FUNCTION_BLOCK xPPU_Crane
VAR_INPUT
	i_error: POINTER TO ErrorManager;
	i_process: POINTER TO ProcessManager;
	i_state: POINTER TO StateTracker;
END_VAR
VAR
	m_emptyParams: ParameterSet;
	m_subRes: EOperationResult;
	m_alarm_flags: ARRAY [1..10] OF BOOL := [FALSE, FALSE, FALSE, FALSE, FALSE, FALSE,FALSE, FALSE, FALSE, FALSE]; 
	m_timer_LSC_EntryCheck : TON;
END_VAR

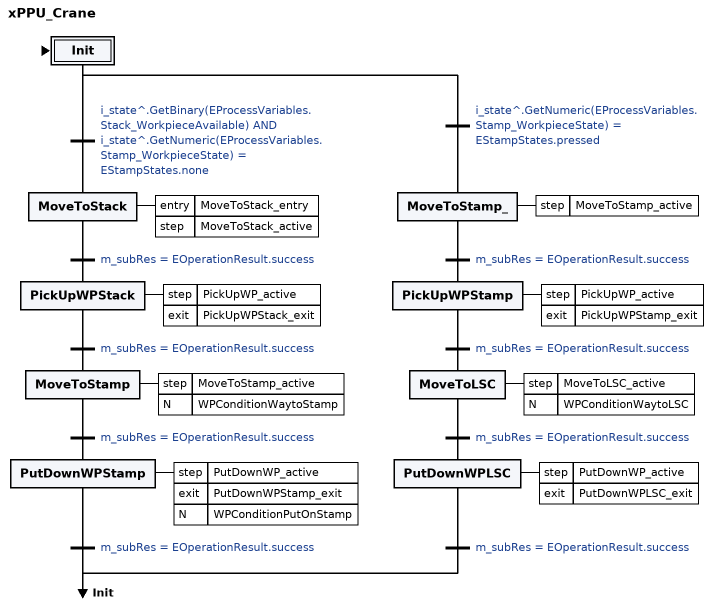
INITIAL_STEP Init:
END_STEP
TRANSITION FROM Init TO MoveToStack
    := i_state^.GetBinary(EProcessVariables.Stack_WorkpieceAvailable) AND i_state^.GetNumeric(EProcessVariables.Stamp_WorkpieceState) = EStampStates.none;
END_TRANSITION
STEP MoveToStack:
    MoveToStack_entry(P1);  // entry action
    MoveToStack_active(N);  // step action
END_STEP
TRANSITION FROM MoveToStack TO PickUpWPStack
    := m_subRes = EOperationResult.success;
END_TRANSITION
STEP PickUpWPStack:
    PickUpWP_active(N);  // step action
    PickUpWPStack_exit(P0);  // exit action
END_STEP
TRANSITION FROM PickUpWPStack TO MoveToStamp
    := m_subRes = EOperationResult.success;
END_TRANSITION
STEP MoveToStamp:
    MoveToStamp_active(N);  // step action
    WPConditionWaytoStamp(N);
END_STEP
TRANSITION FROM MoveToStamp TO PutDownWPStamp
    := m_subRes = EOperationResult.success;
END_TRANSITION
STEP PutDownWPStamp:
    PutDownWP_active(N);  // step action
    PutDownWPStamp_exit(P0);  // exit action
    WPConditionPutOnStamp(N);
END_STEP
TRANSITION FROM PutDownWPStamp TO Init
    := m_subRes = EOperationResult.success;
END_TRANSITION
TRANSITION FROM Init TO MoveToStamp_
    := i_state^.GetNumeric(EProcessVariables.Stamp_WorkpieceState) = EStampStates.pressed;
END_TRANSITION
STEP MoveToStamp_:
    MoveToStamp_active(N);  // step action
END_STEP
TRANSITION FROM MoveToStamp_ TO PickUpWPStamp
    := m_subRes = EOperationResult.success;
END_TRANSITION
STEP PickUpWPStamp:
    PickUpWP_active(N);  // step action
    PickUpWPStamp_exit(P0);  // exit action
END_STEP
TRANSITION FROM PickUpWPStamp TO MoveToLSC
    := m_subRes = EOperationResult.success;
END_TRANSITION
STEP MoveToLSC:
    MoveToLSC_active(N);  // step action
    WPConditionWaytoLSC(N);
END_STEP
TRANSITION FROM MoveToLSC TO PutDownWPLSC
    := m_subRes = EOperationResult.success;
END_TRANSITION
STEP PutDownWPLSC:
    PutDownWP_active(N);  // step action
    PutDownWPLSC_exit(P0);  // exit action
END_STEP
TRANSITION FROM PutDownWPLSC TO Init
    := m_subRes = EOperationResult.success;
END_TRANSITION

ACTION MoveToLSC_active:
m_subRes := i_process^.Execute(
	EBehaviorType.control_primitive,
	EPrimitives.Crane_MoveToLSC,
	m_emptyParams);
END_ACTION

ACTION MoveToStack_active:
m_subRes := i_process^.Execute(
	EBehaviorType.control_primitive,
	EPrimitives.Crane_MoveToStack,
	m_emptyParams);
END_ACTION

ACTION MoveToStack_entry:

END_ACTION

ACTION MoveToStamp_active:
m_subRes := i_process^.Execute(
	EBehaviorType.control_primitive,
	EPrimitives.Crane_MoveToStamp,
	m_emptyParams);
END_ACTION

ACTION PickUpWP_active:
m_subRes := i_process^.Execute(
	EBehaviorType.control_primitive,
	EPrimitives.Crane_PickUpWP,
	m_emptyParams);
END_ACTION

ACTION PickUpWPStack_exit:
i_state^.ShiftProduct(EProducts.stack_product, EProducts.crane_product); 
IF m_alarm_flags[1] = FALSE
	AND i_state^.GetBinary(EProcessVariables.Crane_AtStack)
    AND i_state^.GetBinary(EProcessVariables.Stack_WorkpieceAvailable)
    AND NOT i_state^.GetBinary(EProcessVariables.Crane_HoldingWorkpiece)
THEN 
    i_error^.AddMessage(EAlarms.crane_gripper_failed_stack, TRUE, ESeverity.error, 'Crane failed to pick up the WP at Stack');
    m_alarm_flags[1] := TRUE;
END_IF

IF m_alarm_flags[2] = FALSE
	AND i_state^.GetBinary(EProcessVariables.Crane_AtStack)
    AND NOT i_state^.GetBinary(EProcessVariables.Stack_WorkpieceAvailable) 
    AND NOT i_state^.GetBinary(EProcessVariables.Crane_HoldingWorkpiece)
THEN 
    i_error^.AddMessage(EAlarms.crane_dropped_WP_stack, TRUE, ESeverity.error, 'WP dropped from Crane at Stack');
    m_alarm_flags[2] := TRUE;
END_IF
END_ACTION

ACTION PickUpWPStamp_exit:
i_state^.ShiftProduct(EProducts.stamp_product, EProducts.crane_product);
IF m_alarm_flags[5] = FALSE
    AND i_state^.GetBinary(EProcessVariables.Crane_AtStamp) 
    AND NOT i_state^.GetBinary(EProcessVariables.Crane_HoldingWorkpiece)
	AND i_state^.GetBinary(EProcessVariables.Stamp_WPAtStamp)
THEN 
    i_error^.AddMessage(EAlarms.crane_gripper_failed_stamp, TRUE, ESeverity.error, 'Crane failed pick the WP up at Stamp');
    m_alarm_flags[5] := TRUE;
END_IF

IF m_alarm_flags[6] = FALSE
    AND i_state^.GetBinary(EProcessVariables.Crane_AtStamp) 
    AND NOT i_state^.GetBinary(EProcessVariables.Crane_HoldingWorkpiece)
	AND NOT i_state^.GetBinary(EProcessVariables.Stamp_WPAtStamp)
THEN 
    i_error^.AddMessage(EAlarms.crane_dropped_WP_stamp, TRUE, ESeverity.error, 'WP dropped from Crane at Stamp');
    m_alarm_flags[6] := TRUE;
END_IF
END_ACTION

ACTION PutDownWP_active:
m_subRes := i_process^.Execute(
	EBehaviorType.control_primitive,
	EPrimitives.Crane_PutDownWP,
	m_emptyParams);
END_ACTION

ACTION PutDownWPLSC_exit:
i_state^.ShiftProduct(EProducts.crane_product, EProducts.LSC_product);
END_ACTION

ACTION PutDownWPStamp_exit:
i_state^.ShiftProduct(EProducts.crane_product, EProducts.stamp_product);
END_ACTION

ACTION WPConditionPutOnStamp:
IF m_alarm_flags[4] = FALSE
	AND i_state^.Getbinary(EProcessVariables.Crane_AtStamp)
    AND i_state^.Getbinary(EProcessVariables.Crane_CylinderExtended)
	AND NOT i_state^.Getbinary(EProcessVariables.Stamp_WPAtStamp)
THEN 
    i_error^.AddMessage(EAlarms.crane_putdown_failed_stamp, TRUE, ESeverity.error, 'WP not corrcetly put by the Crane at Stamp');
    m_alarm_flags[4] := TRUE;
END_IF
END_ACTION

ACTION WPConditionWaytoLSC:
IF m_alarm_flags[7] = FALSE
    AND NOT i_state^.GetBinary(EProcessVariables.Crane_HoldingWorkpiece)
THEN 
    i_error^.AddMessage(EAlarms.crane_dropped_WP_WayToLSC, TRUE, ESeverity.error, 'WP dropped from Crane on the way to LSC');
    m_alarm_flags[7] := TRUE;
END_IF
END_ACTION

ACTION WPConditionWaytoStamp:
IF m_alarm_flags[3] = FALSE
    AND NOT i_state^.GetBinary(EProcessVariables.Crane_HoldingWorkpiece)
THEN 
    i_error^.AddMessage(EAlarms.crane_dropped_WP_WayToStamp, TRUE, ESeverity.error, 'WP dropped from Crane on the way to Stamp');
    m_alarm_flags[3] := TRUE;
END_IF
END_ACTION

END_FUNCTION_BLOCK

(* stored: Version 1.1.0.1
   POU xPPU_Crane: Id {78161606-71b4-4291-9ac3-095c552c2798}, SpecialFunc None
   Action MoveToLSC_active: Id {8277d77e-cd34-4ec5-9f75-b93467ba1bb6}
   Action MoveToStack_active: Id {571b406f-6c8e-4544-9ae9-49953b6b39be}
   Action MoveToStack_entry: Id {ce2a418a-1861-4bd8-b286-83f8f539ccb0}
   Action MoveToStamp_active: Id {a7848926-ee25-41bb-a037-2f10498f3c62}
   Action PickUpWP_active: Id {0442f4fd-88ed-4177-bc1f-6efb591dfd4d}
   Action PickUpWPStack_exit: Id {1b736f68-d7a0-4bc6-af85-9b732ac83761}
   Action PickUpWPStamp_exit: Id {6d99610e-69d1-409d-88f0-202e27f184fb}
   Action PutDownWP_active: Id {c713f15e-67e6-4a12-b1c1-93deb7666c90}
   Action PutDownWPLSC_exit: Id {f398bd84-d715-4628-8579-139e0657ea82}
   Action PutDownWPStamp_exit: Id {39d022ad-1212-45a5-b9d2-c0ff009b69d4}
   Action WPConditionPutOnStamp: Id {8c333206-6540-47ac-8fcb-1788ac4128fa}
   Action WPConditionWaytoLSC: Id {288de139-2c26-4df1-97af-b3a9016fcd87}
   Action WPConditionWaytoStamp: Id {e4adebe5-6f6b-476d-b387-4f8235d3d30a} *)
